PROGRAM INTERNAL PRG_TEST_FB_LOGGER
VAR
	fbLogHandler_TxtFile :	FB_LogHandler_TxtFile(
									sLogFolder := 'D:\Temp\',
									sLogFilePrefix := 'AutomaticTestLog_',
									sLogFileExtension := 'txt',
									nMaxLogFileSize := 500,
									nMaxNumberOfLogFiles := 3
								);
	fbLogger : FB_Logger;
	bEnableTests : BOOL;
	bAddToLog : BOOL;
	bStressTest : BOOL;
	nIdx : UDINT;
	sMsg : T_MaxString;
END_VAR

IF bEnableTests THEN
	fbLogger.AddLogHandler(fbLogHandler_TxtFile);
	fbLogger.Run();
	IF bAddToLog THEN
		bAddToLog := FALSE;
		fbLogger.DEBUG(sMsg);
	END_IF
	IF bStressTest THEN
		// Write an item to the log every PLC cycle, this should trigger a buffer overflow
		nIdx := nIdx + 1;
		sMsg := UDINT_TO_STRING(nIdx);
		fbLogger.DEBUG(sMsg);
	END_IF
END_IF

END_PROGRAM

(* stored: Version 1.1.0.1, ProductVersion 3.1.4024.11
   POU PRG_TEST_FB_LOGGER: Id {90bc222e-4655-0939-07a6-64349ec214b9}, SpecialFunc None *)
